TYPE ST_Frame :
STRUCT
	m_pos :ARRAY [1..3] OF LREAL:=[0, 0, 0];
	m_rot :ARRAY[1..3,1..3] OF LREAL:=[1, 0, 0, 0, 1, 0, 0, 0, 1];
END_STRUCT
END_TYPE

(* stored: Version 1.1.0.1, ProductVersion 3.1.4024.12
   DUT ST_Frame: Id {0c0aabb6-6c60-4edd-80ca-fa032ce1cbfa} *)
